// Annex A/B pattern on the base class: the type is ONLY its device logic.
FUNCTION_BLOCK FB_CylinderCM EXTENDS FB_ControlModuleBase
VAR_INPUT
    Command : E_CylinderCommand;
    ParCfg : ST_CylinderParCfg;
    ParCmd : ST_CylinderParCmd;
END_VAR
VAR_OUTPUT
    OutCmd : ST_CylinderOutCmd;
    OutImm : ST_CylinderOutImm;
    Intlk  : FB_PermIntlk;
END_VAR
VAR
    {attribute 'OPC.UA.DA' := '0'}
    _hal    : REFERENCE TO ST_CylinderHal;
    {attribute 'OPC.UA.DA' := '0'}
    _recipe : I_RecipeProvider;
    _tMove  : TON;
    _areaSafe : BOOL := TRUE;           // §7.2 application-supplied area/process interlock
    _areaSafeKey : STRING(255);
    _parCfgStaged : ST_CylinderParCfg;
    _recipePrepared : BOOL;
    _directionPermitsConfigured : BOOL;
    _extendPermit, _retractPermit : BOOL := TRUE;
    _extendPermitKey, _retractPermitKey : STRING(255);
    _extendedSensorTag, _retractedSensorTag : STRING(80);
    _extendedSensorAddress, _retractedSensorAddress : STRING(80);
    _extendOutputTag, _retractOutputTag : STRING(80);
    _extendedTimeoutKey, _retractedTimeoutKey, _bothSensorsKey : STRING(255);
    _bothSensorTags, _bothSensorAddresses : STRING(80);
END_VAR

Cyclic();

METHOD PROTECTED OnCyclic : DINT
OnCyclic := SUPER^.OnCyclic();
Intlk.Cond[1] := _areaSafe;             // §7.2 area-safe/air-ok, supplied via SetAreaSafe
IF NOT _directionPermitsConfigured OR (Command = E_CylinderCommand.NONE) THEN
    Intlk.Cond[2] := TRUE;
ELSIF Command = E_CylinderCommand.EXTEND THEN
    Intlk.Cond[2] := _extendPermit;
ELSIF Command = E_CylinderCommand.RETRACT THEN
    Intlk.Cond[2] := _retractPermit;
ELSE
    Intlk.Cond[2] := FALSE;
END_IF
Intlk();
IF __ISVALIDREF(_hal) THEN              // defensive (§5.6) [TC3]
    OutImm.Extended  := _hal.ExtendedFb;
    OutImm.Retracted := _hal.RetractedFb;
END_IF
OutImm.ExtendedSensorTag := _extendedSensorTag;
OutImm.RetractedSensorTag := _retractedSensorTag;
OutImm.ExtendOutputTag := _extendOutputTag;
OutImm.RetractOutputTag := _retractOutputTag;
OutImm.Diagnostic := Status.Diagnostic;
END_METHOD

// Schematic identity is application configuration, not device behavior.
// Diagnostics keep SourcePath as this module and add the exact failed channel.
METHOD ConfigureIoIdentity
VAR_INPUT
    Identity : ST_CylinderIoIdentity;
END_VAR
_extendedSensorTag := Identity.ExtendedSensor.Tag;
_extendedSensorAddress := Identity.ExtendedSensor.Address;
_retractedSensorTag := Identity.RetractedSensor.Tag;
_retractedSensorAddress := Identity.RetractedSensor.Address;
_extendOutputTag := Identity.ExtendOutput.Tag;
_retractOutputTag := Identity.RetractOutput.Tag;
_extendedTimeoutKey := Identity.ExtendedTimeoutKey;
_retractedTimeoutKey := Identity.RetractedTimeoutKey;
_bothSensorsKey := Identity.BothSensorsKey;
_bothSensorTags := CONCAT(Identity.ExtendedSensor.Tag, CONCAT(' / ', Identity.RetractedSensor.Tag));
_bothSensorAddresses := CONCAT(Identity.ExtendedSensor.Address, CONCAT(' / ', Identity.RetractedSensor.Address));
END_METHOD

// Functional stop used by an owning sequence on abort/interlock loss.
// This is not a certified stop; the safety system remains authoritative.
METHOD WithdrawOutputs
IF __ISVALIDREF(_hal) THEN
    _hal.ExtendOut := FALSE;
    _hal.RetractOut := FALSE;
END_IF
END_METHOD

// Symmetric counterpart to WithdrawOutputs, for an owning sequence that withdrew a
// cylinder to hold a phase and now wants it driving again — a press dwell whose
// two-hand button was released and re-pressed, where the force comes from the valve
// latched by the already-completed EXTEND, so nothing else would re-energize it.
// Re-asserts ONLY the last commanded direction and ONLY while that direction's own
// permit is satisfied, so it can never restore an output the interlock is withholding:
// the caller asks, this module still decides. Idempotent; safe to call every scan.
// Not a certified enable — the safety system remains authoritative (§9).
METHOD RestoreOutputs
VAR
    permitted : BOOL;
END_VAR
IF NOT __ISVALIDREF(_hal) THEN
    RETURN;
END_IF
IF Command = E_CylinderCommand.EXTEND THEN
    permitted := _extendPermit OR NOT _directionPermitsConfigured;
ELSIF Command = E_CylinderCommand.RETRACT THEN
    permitted := _retractPermit OR NOT _directionPermitsConfigured;
ELSE
    permitted := FALSE;                 // no direction commanded: nothing to restore (§5.6)
END_IF
IF NOT permitted OR NOT Intlk.AllOk THEN
    RETURN;
END_IF
_hal.ExtendOut  := (Command = E_CylinderCommand.EXTEND);
_hal.RetractOut := (Command = E_CylinderCommand.RETRACT);
END_METHOD

METHOD PROTECTED OnAbort : DINT
OnAbort := SUPER^.OnAbort();            // base first (§3.14.2)
IF __ISVALIDREF(_hal) THEN
    _hal.ExtendOut := FALSE;
    _hal.RetractOut := FALSE;
END_IF
END_METHOD

METHOD PrepareRecipe : BOOL
VAR_INPUT
    Model : ST_ModelId;
END_VAR
IF _recipe = 0 THEN
    _parCfgStaged := ParCfg;
    _recipePrepared := TRUE;
    PrepareRecipe := TRUE;
ELSIF _recipe.Load(ModelCode := Model.ModelCode, RecipeKey := 'CylinderCM', pParCfg := ADR(_parCfgStaged), Size := SIZEOF(_parCfgStaged)) THEN
    _recipePrepared := TRUE;
    PrepareRecipe := TRUE;
ELSE
    _M_Fault(E_Reason.RECIPE_INVALID, 'std.error.recipeSchemaInvalid');
    _recipePrepared := FALSE;
    PrepareRecipe := FALSE;
END_IF
END_METHOD

METHOD CommitRecipe
IF _recipePrepared THEN ParCfg := _parCfgStaged; END_IF
_recipePrepared := FALSE;
END_METHOD

METHOD AbortRecipe
_recipePrepared := FALSE;
END_METHOD

METHOD Setup : BOOL
VAR_INPUT
    Name   : STRING(80);
    HalRef : REFERENCE TO ST_CylinderHal;
    Recipe : I_RecipeProvider;
END_VAR
VAR
    InitialModel : ST_ModelId;
END_VAR
_M_SetName(Name);
_M_SetPresentation(DisplayNameKey := 'std.moduleType.cylinder.name', DescriptionKey := 'std.moduleType.cylinder.description', TypeKey := 'std.moduleType.cylinder');
_hal REF= HalRef;                        // [TC3] TC3 §3.11
_recipe := Recipe;
// A library type owns a std.* key; an application overrides the text through
// SetAreaSafe when its own condition is more specific (§7.2.1).
Intlk.Define(Index := 1, Description := 'std.interlock.areaSafe', Reason := E_Reason.INTERLOCK_DROPPED, Bypassable := FALSE);
Intlk.Define(Index := 2, Description := 'std.interlock.directionPermitted', Reason := E_Reason.INTERLOCK_DROPPED, Bypassable := FALSE);
_M_PublishCommand(Value := TO_DINT(E_CylinderCommand.EXTEND), Label := 'std.command.extend');
_M_PublishCommand(Value := TO_DINT(E_CylinderCommand.RETRACT), Label := 'std.command.retract');
Setup := PrepareRecipe(Model := InitialModel);
IF Setup THEN CommitRecipe(); END_IF
END_METHOD

// Core §7.2/§7.2.1 — the application supplies this type's area/process interlock,
// the same shape as SetDirectionalPermits: a method (not an OPC UA write), and the
// condition is re-evaluated every scan so a manual command obeys the same rule.
//
// This replaces a SIM-only force hook that used to drive Cond[1] directly. That
// hook was the ONLY writer of the condition, so the slot an operator sees as
// "area safe" could be moved by a test and by nothing else: a reusable type
// published an interlock its application had no way to supply (§7.2.1), and the
// bypass shipped in every release build (§5.7). Driving the real condition is
// also strictly better test evidence - T3 now exercises the shipped path.
//
// Defaults TRUE: a station that declares no area interlock is not gated by one.
METHOD SetAreaSafe
VAR_INPUT
    Ok : BOOL;
    DescriptionKey : STRING(255);
END_VAR
_areaSafe := Ok;
_areaSafeKey := DescriptionKey;
IF _areaSafeKey <> '' THEN
    Intlk.Define(Index := 1, Description := _areaSafeKey, Reason := E_Reason.INTERLOCK_DROPPED, Bypassable := FALSE);
ELSE
    ;
END_IF
END_METHOD

METHOD PROTECTED _M_Dispatch
VAR
    ext : BOOL;
    d   : ST_Diagnostic;
END_VAR
IF _manualReq THEN
    _manualReq := FALSE;
    IF (_manualCmd = TO_DINT(E_CylinderCommand.EXTEND)) OR (_manualCmd = TO_DINT(E_CylinderCommand.RETRACT)) THEN
        Command := _manualCmd;
    ELSE
        _M_Fault(E_Reason.UNSUPPORTED_COMMAND, 'std.error.unsupportedCylinderCommand');
        RETURN;
    END_IF
END_IF
IF (Command <> E_CylinderCommand.EXTEND) AND (Command <> E_CylinderCommand.RETRACT) THEN
    _M_Fault(E_Reason.UNSUPPORTED_COMMAND, 'std.error.unsupportedCylinderCommand');
    RETURN;
END_IF
IF Command = E_CylinderCommand.EXTEND THEN
    _M_TagCommand(Id := 1, Label := 'std.command.extend');       // §8.11.4(a)
    IF _directionPermitsConfigured THEN
        Intlk.Define(Index := 2, Description := _extendPermitKey, Reason := E_Reason.INTERLOCK_DROPPED, Bypassable := FALSE);
        Intlk.Cond[2] := _extendPermit;
    ELSE
        Intlk.Cond[2] := TRUE;
    END_IF
ELSE
    _M_TagCommand(Id := 2, Label := 'std.command.retract');
    IF _directionPermitsConfigured THEN
        Intlk.Define(Index := 2, Description := _retractPermitKey, Reason := E_Reason.INTERLOCK_DROPPED, Bypassable := FALSE);
        Intlk.Cond[2] := _retractPermit;
    ELSE
        Intlk.Cond[2] := TRUE;
    END_IF
END_IF
Intlk();
IF NOT Intlk.AllOk THEN
    // §6.1 HELD, not a fault. An interlock is by definition a condition that must
    // hold DURING motion, and losing one is often expected operator behaviour —
    // releasing a two-hand button is the designed way to stop a stroke. Faulting
    // classified that as a defect and forced the ABORTED/STOPPED exit (Reset ->
    // IDLE), which on the press was unreachable: the fault's own condition included
    // "two-hand held during a stroke", which can only be restored by running.
    // Nothing is weakened here — the output is withdrawn in the same place, by the
    // same permit — only the classification and the way out change: the module stays
    // BUSY with its outputs off and resumes when the condition returns (§8.4: this
    // is a wait, not a downtime event). Rewinding to N010 means the resume
    // re-energizes the direction output and re-arms MoveTimeout with a full window,
    // so a hold cannot silently consume the travel time it was not moving for.
    _hal.ExtendOut := FALSE;
    _hal.RetractOut := FALSE;
    d := Intlk.Diagnostic;
    d.SourcePath := _name;                            // owner sets the path (§7.2)
    _M_HoldDiag(Diag := d);
    _step := 10;
    RETURN;
END_IF
IF _hal.ExtendedFb AND _hal.RetractedFb THEN
    IF _bothSensorsKey <> '' THEN
        _M_FaultIoN(Code := PL_ModuleReasons.CYL_BOTH_SENSORS, Text := _bothSensorsKey,
            IoTag := _bothSensorTags, IoAddress := _bothSensorAddresses);
    ELSE
        _M_FaultN(Code := PL_ModuleReasons.CYL_BOTH_SENSORS, Text := 'std.error.cylinderBothSensors');
    END_IF
    RETURN;
END_IF
ext := (Command = E_CylinderCommand.EXTEND);
CASE _step OF
    10:
        OutCmd.Reached := FALSE;
        _hal.ExtendOut  := ext;
        _hal.RetractOut := NOT ext;
        _tMove(IN := FALSE);
        _step := 20;
    20:
        _tMove(IN := TRUE, PT := ParCfg.MoveTimeout);
        IF (ext AND _hal.ExtendedFb) OR ((NOT ext) AND _hal.RetractedFb) THEN
            _tMove(IN := FALSE);
            OutCmd.Reached := TRUE;
            _M_Complete();
        ELSIF _tMove.Q THEN
            _tMove(IN := FALSE);
            IF ext AND (_extendedSensorTag <> '') THEN
                _M_FaultIoN(Code := PL_ModuleReasons.CYL_NOT_EXTENDED, Text := _extendedTimeoutKey,
                    IoTag := _extendedSensorTag, IoAddress := _extendedSensorAddress);
            ELSIF (NOT ext) AND (_retractedSensorTag <> '') THEN
                _M_FaultIoN(Code := PL_ModuleReasons.CYL_NOT_RETRACTED, Text := _retractedTimeoutKey,
                    IoTag := _retractedSensorTag, IoAddress := _retractedSensorAddress);
            ELSIF ext THEN
                _M_FaultN(Code := PL_ModuleReasons.CYL_NOT_EXTENDED, Text := 'std.error.cylinderExtendTimeout');
            ELSE
                _M_FaultN(Code := PL_ModuleReasons.CYL_NOT_RETRACTED, Text := 'std.error.cylinderRetractTimeout');
            END_IF
        END_IF
ELSE
    _M_Fault(E_Reason.STEP_STALLED, 'std.error.undefinedStep');    // defined ELSE (§5.6)
END_CASE
END_METHOD

// Functional collision/process interlocks supplied by the owning EM/Unit.
// Methods are not OPC UA writes; the check is repeated inside dispatch so manual
// commands use the same rule. Certified safety remains external.
METHOD SetDirectionalPermits
VAR_INPUT
    ExtendOk : BOOL;
    RetractOk : BOOL;
    ExtendDescriptionKey : STRING(255);
    RetractDescriptionKey : STRING(255);
END_VAR
_directionPermitsConfigured := TRUE;
_extendPermit := ExtendOk;
_retractPermit := RetractOk;
_extendPermitKey := ExtendDescriptionKey;
_retractPermitKey := RetractDescriptionKey;
END_METHOD

// Pure release-query companion to SetDirectionalPermits. The owning Unit uses
// this for act-or-explain so the HMI checks the exact permit used by dispatch.
METHOD AppendDirectionalRelease : INT
VAR_INPUT
    Value : DINT;
END_VAR
VAR_IN_OUT
    Report : ST_ReleaseReport;
END_VAR
VAR
    permitted : BOOL;
    validCommand : BOOL;
    descriptionKey : STRING(255);
END_VAR
permitted := TRUE;
validCommand := (Value = TO_DINT(E_CylinderCommand.EXTEND))
    OR (Value = TO_DINT(E_CylinderCommand.RETRACT));
descriptionKey := '';
IF _directionPermitsConfigured AND (Value = TO_DINT(E_CylinderCommand.EXTEND)) THEN
    permitted := _extendPermit;
    descriptionKey := _extendPermitKey;
ELSIF _directionPermitsConfigured AND (Value = TO_DINT(E_CylinderCommand.RETRACT)) THEN
    permitted := _retractPermit;
    descriptionKey := _retractPermitKey;
ELSIF NOT validCommand THEN
    permitted := FALSE;
    descriptionKey := 'std.error.unsupportedCylinderCommand';
ELSE
    permitted := TRUE;
END_IF
IF NOT permitted AND (Report.Count < PL_Fraktal.MAX_RELEASE_REASONS) THEN
    Report.Count := Report.Count + 1;
    Report.Reasons[Report.Count].Description := descriptionKey;
    Report.Reasons[Report.Count].SourcePath := _name;
    IF validCommand THEN
        Report.Reasons[Report.Count].ReasonCode := E_Reason.INTERLOCK_DROPPED;
    ELSE
        Report.Reasons[Report.Count].ReasonCode := E_Reason.UNSUPPORTED_COMMAND;
    END_IF
    Report.Reasons[Report.Count].Kind := E_ReleaseKind.INTERLOCK;
    Report.Reasons[Report.Count].Bypassable := FALSE;
END_IF
AppendDirectionalRelease := Report.Count;
END_METHOD

METHOD PROTECTED _M_PublishStatus
SUPER^._M_PublishStatus();
OutImm.Diagnostic := Status.Diagnostic;
END_METHOD

END_FUNCTION_BLOCK

(* stored: Version 1.1.0.1, ProductVersion 3.1.4024.12
   POU FB_CylinderCM: Id {05f548d6-e819-40c3-b0bd-f2c5ee607509}, SpecialFunc None
   Method OnCyclic: Id {d8d68e4c-1628-4704-abda-c173c26a6684}
   Method ConfigureIoIdentity: Id {da966427-aa84-430d-aaaf-6b2d28cf8331}
   Method WithdrawOutputs: Id {4d586967-b1ec-46e2-b210-b0d4c6f593a0}
   Method RestoreOutputs: Id {a9daf69a-0e65-485d-8e32-c25880649db8}
   Method OnAbort: Id {e057e446-dbf0-4d4e-8095-e77cb11fc9d8}
   Method PrepareRecipe: Id {9fc6da18-1a34-436f-b95f-8a202c41c2f2}
   Method CommitRecipe: Id {2507146c-6bb3-4103-92db-e1e95f4c558c}
   Method AbortRecipe: Id {56e645a8-70e5-4384-88bd-bbc05886f071}
   Method Setup: Id {4aaae498-7dfe-4e4f-b767-65724d335fde}
   Method SetAreaSafe: Id {d171827b-01bb-4ec3-82bc-76f0b19118b9}
   Method _M_Dispatch: Id {f4246abc-e03f-4d9d-9774-cf8b297a7d67}
   Method SetDirectionalPermits: Id {b1045a9a-9497-4b07-b315-d6be9086fd4c}
   Method AppendDirectionalRelease: Id {13e02c3d-0e9d-4f2f-8820-1b10fc328401}
   Method _M_PublishStatus: Id {014aa002-cf47-48a0-96b5-ed59efddfa57} *)
